// TIA Portal project "Auto Jollof Rice Cooker" (V15.1)
// This is built as a first time project and it is simulated independently to show how pneumatic machines operates.

(* hardware
DEVICE "S7-1200 station_1"  S7-1200 Station
   slot 0: "Rack_0"  S7-1200 Rack  Rack  V1.0
   slot 1: "PLC_1"  CPU 1212FC DC/DC/RLY  6ES7 212-1HF40-0XB0  V4.2
*)

// ===== PLC "PLC_1"  CPU 1212FC DC/DC/RLY =====

VAR_GLOBAL   // PLC tag table "Default tag table"
   "Start_Button" AT %M0.0 : Bool;
   "rice_cooker" AT %M0.1 : Bool;
   "water_nozzle" AT %M0.2 : Bool;
   "ingredient1_nozzle" AT %M0.3 : Bool;
   "ingredient2_nozzle" AT %M0.4 : Bool;
   "frying_oven" AT %M0.5 : Bool;
   "groundnut_oil" AT %M0.6 : Bool;
   "light_fry_mode" AT %M0.7 : Bool;
   "deep_fry_mode" AT %M1.0 : Bool;
   "alarm" AT %M1.1 : Bool;
   "vending_area" AT %M1.2 : Bool;
   "dispense_butoon" AT %M1.3 : Bool;
   "thank_you_message" AT %M1.4 : Bool;
   "phase2_start" AT %M1.5 : Bool;
   "phase3_start" AT %M1.6 : Bool;
   "phase4 start" AT %M1.7 : Bool;
   "phase5_start" AT %M2.0 : Bool;
   "phase6_start" AT %M2.1 : Bool;
   "phase7_start" AT %M2.2 : Bool;
   "cycle_done" AT %M2.3 : Bool;
END_VAR

VAR_GLOBAL CONSTANT   // PLC tag table "Default tag table"
   "water_nozzle_timer" : Time := T#10s;
   "ingredient1_nozzle_timer" : Time := T#1s;
   "ingredient2_nozzle_timer" : Time := T#5s;
   "countdown_vending_phase_timer" : Time := T#120s;
END_VAR

// folder: System blocks/Program resources

DATA_BLOCK "countdown water nozzle"   // DB1
{ S7_Optimized_Access := 'TRUE' }
AUTHOR : Simatic
FAMILY : IEC
NAME : IEC_TMR
VERSION : 1.0
// stored: InstanceOfName IEC_TIMER
"IEC_TIMER"
BEGIN
END_DATA_BLOCK

DATA_BLOCK "Time water nozzle stay ON"   // DB2
{ S7_Optimized_Access := 'TRUE' }
AUTHOR : Simatic
FAMILY : IEC
NAME : IEC_TMR
VERSION : 1.0
// stored: InstanceOfName IEC_TIMER
"IEC_TIMER"
BEGIN
END_DATA_BLOCK

DATA_BLOCK "Countdown Ingredient 1"   // DB3
{ S7_Optimized_Access := 'TRUE' }
AUTHOR : Simatic
FAMILY : IEC
NAME : IEC_TMR
VERSION : 1.0
// stored: InstanceOfName IEC_TIMER
"IEC_TIMER"
BEGIN
END_DATA_BLOCK

DATA_BLOCK "to count the process for five times then stop"   // DB4
{ S7_Optimized_Access := 'TRUE' }
AUTHOR : Simatic
FAMILY : IEC
NAME : CNTR
VERSION : 1.0
// stored: InstanceOfName IEC_COUNTER
"IEC_COUNTER"
BEGIN
END_DATA_BLOCK

DATA_BLOCK "Time Ingredient 1 Nozzle Stays ON"   // DB5
{ S7_Optimized_Access := 'TRUE' }
AUTHOR : Simatic
FAMILY : IEC
NAME : IEC_TMR
VERSION : 1.0
// stored: InstanceOfName IEC_TIMER
"IEC_TIMER"
BEGIN
END_DATA_BLOCK

DATA_BLOCK "Countdown Ingredient 2"   // DB6
{ S7_Optimized_Access := 'TRUE' }
AUTHOR : Simatic
FAMILY : IEC
NAME : IEC_TMR
VERSION : 1.0
// stored: InstanceOfName IEC_TIMER
"IEC_TIMER"
BEGIN
END_DATA_BLOCK

DATA_BLOCK "Time Ingredient 2 Nozzle Stays ON"   // DB7
{ S7_Optimized_Access := 'TRUE' }
AUTHOR : Simatic
FAMILY : IEC
NAME : IEC_TMR
VERSION : 1.0
// stored: InstanceOfName IEC_TIMER
"IEC_TIMER"
BEGIN
END_DATA_BLOCK

DATA_BLOCK "Countdown Frying Phase"   // DB8
{ S7_Optimized_Access := 'TRUE' }
AUTHOR : Simatic
FAMILY : IEC
NAME : IEC_TMR
VERSION : 1.0
// stored: InstanceOfName IEC_TIMER
"IEC_TIMER"
BEGIN
END_DATA_BLOCK

DATA_BLOCK "Countdown Groundnut OIl ON"   // DB9
{ S7_Optimized_Access := 'TRUE' }
AUTHOR : Simatic
FAMILY : IEC
NAME : IEC_TMR
VERSION : 1.0
// stored: InstanceOfName IEC_TIMER
"IEC_TIMER"
BEGIN
END_DATA_BLOCK

DATA_BLOCK "G.OIl stay ON Timer"   // DB10
{ S7_Optimized_Access := 'TRUE' }
AUTHOR : Simatic
FAMILY : IEC
NAME : IEC_TMR
VERSION : 1.0
// stored: InstanceOfName IEC_TIMER
"IEC_TIMER"
BEGIN
END_DATA_BLOCK

DATA_BLOCK "Countdown Vending Start"   // DB11
{ S7_Optimized_Access := 'TRUE' }
AUTHOR : Simatic
FAMILY : IEC
NAME : IEC_TMR
VERSION : 1.0
// stored: InstanceOfName IEC_TIMER
"IEC_TIMER"
BEGIN
END_DATA_BLOCK

DATA_BLOCK "Fring Oven stays ON Timer"   // DB12
{ S7_Optimized_Access := 'TRUE' }
AUTHOR : Simatic
FAMILY : IEC
NAME : IEC_TMR
VERSION : 1.0
// stored: InstanceOfName IEC_TIMER
"IEC_TIMER"
BEGIN
END_DATA_BLOCK

// folder: (top level)

ORGANIZATION_BLOCK "Main"   // OB1, LAD, ProgramCycle
TITLE = "Main Program Sweep (Cycle)"
{ S7_Optimized_Access := 'TRUE' }
VERSION : 0.1
   VAR_INPUT
      Initial_Call : Bool;   // Initial call of this OB
      Remanence : Bool;   // =True, if remanent data are available
   END_VAR
BEGIN

REGION Network 1
   // phase 1 rice cooker comes ON with parboiled rice already placed on the inbuilt pot.
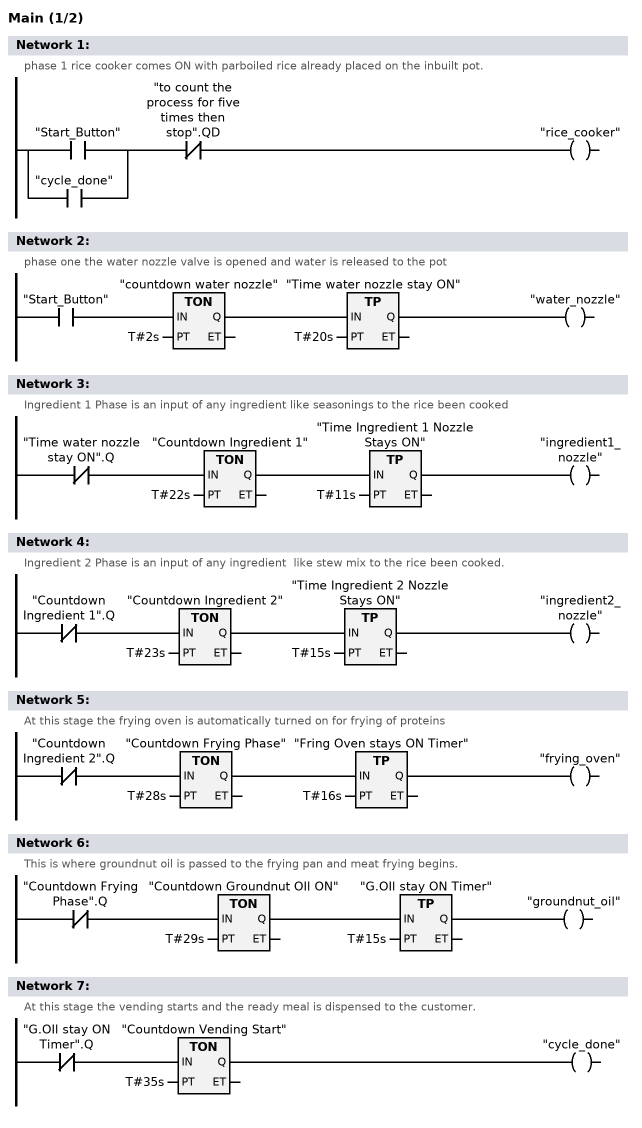
   RUNG wire#powerrail
      Contact( "Start_Button" )
      wire#w1
      I_Contact( "to count the process for five times then stop".QD )
      Coil( "rice_cooker" )
   END_RUNG
   RUNG wire#powerrail
      Contact( "cycle_done" )
   END_RUNG wire#w1
   // the same network as SCL:
   "rice_cooker" := ("Start_Button" OR "cycle_done") AND NOT "to count the process for five times then stop".QD;
END_REGION

REGION Network 2
   // phase one the water nozzle valve is opened and water is released to the pot
   "countdown water nozzle".TON(IN := "Start_Button", PT := T#2s);
   "Time water nozzle stay ON".TP(IN := "countdown water nozzle".Q, PT := T#20s);
   "water_nozzle" := "Time water nozzle stay ON".Q;
END_REGION

REGION Network 3
   // Ingredient 1 Phase is an input of any ingredient like seasonings to the rice been cooked
   "Countdown Ingredient 1".TON(IN := NOT "Time water nozzle stay ON".Q, PT := T#22s);
   "Time Ingredient 1 Nozzle Stays ON".TP(IN := "Countdown Ingredient 1".Q, PT := T#11s);
   "ingredient1_nozzle" := "Time Ingredient 1 Nozzle Stays ON".Q;
END_REGION

REGION Network 4
   // Ingredient 2 Phase is an input of any ingredient  like stew mix to the rice been cooked.
   "Countdown Ingredient 2".TON(IN := NOT "Countdown Ingredient 1".Q, PT := T#23s);
   "Time Ingredient 2 Nozzle Stays ON".TP(IN := "Countdown Ingredient 2".Q, PT := T#15s);
   "ingredient2_nozzle" := "Time Ingredient 2 Nozzle Stays ON".Q;
END_REGION

REGION Network 5
   // At this stage the frying oven is automatically turned on for frying of proteins
   "Countdown Frying Phase".TON(IN := NOT "Countdown Ingredient 2".Q, PT := T#28s);
   "Fring Oven stays ON Timer".TP(IN := "Countdown Frying Phase".Q, PT := T#16s);
   "frying_oven" := "Fring Oven stays ON Timer".Q;
END_REGION

REGION Network 6
   // This is where groundnut oil is passed to the frying pan and meat frying begins.
   "Countdown Groundnut OIl ON".TON(IN := NOT "Countdown Frying Phase".Q, PT := T#29s);
   "G.OIl stay ON Timer".TP(IN := "Countdown Groundnut OIl ON".Q, PT := T#15s);
   "groundnut_oil" := "G.OIl stay ON Timer".Q;
END_REGION

REGION Network 7
   // At this stage the vending starts and the ready meal is dispensed to the customer.
   "Countdown Vending Start".TON(IN := NOT "G.OIl stay ON Timer".Q, PT := T#35s);
   "cycle_done" := "Countdown Vending Start".Q;
END_REGION

REGION Network 8
   // We placed an up counter to count the no of times that it cooks per day. and made the total no of times to cook in a day to be 10 times. Once it gets to 10, the start cooking button becomes inactive.
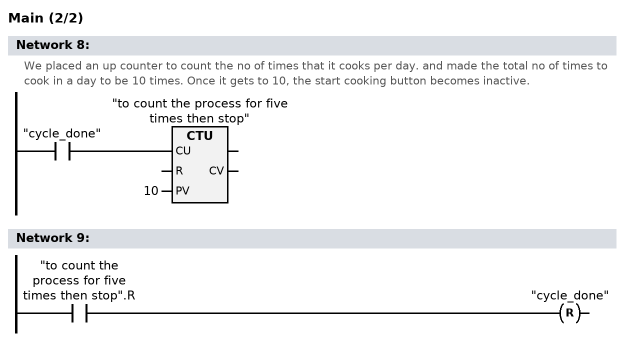
   "to count the process for five times then stop".CTU(CU := "cycle_done", PV := 10);
END_REGION

REGION Network 9
   RUNG wire#powerrail
      Contact( "to count the process for five times then stop".R )
      R_Coil( "cycle_done" )
   END_RUNG
   // the same network as SCL:
   IF "to count the process for five times then stop".R THEN "cycle_done" := FALSE; END_IF;
END_REGION
END_ORGANIZATION_BLOCK